(* IEC 61131-3 sources: T4Exjobb/Sigma/Stations/MachineControl/MachineControl/Class/_SysDateTime2, 1 file *)

(* ---- _SysDateTime2.st ---- *)
(*!
<Class
	Name               = "_SysDateTime2"
	Revision           = "0.0"
	RealtimeTask       = "false"
	CyclicTask         = "false"
	BackgroundTask     = "true"
	DefBackground      = "100 ms"
	Sigmatek           = "true"
	OSInterface        = "false"
	HighPriority       = "false"
	Automatic          = "false"
	UpdateMode         = "Prescan"
	SharedCommandTable = "true"
	Objectsize         = "(284,120)">
	<Channels>
		<Server Name="Day" Visualized="true" Initialize="false" WriteProtected="false" Retentive="false"/>
		<Server Name="Hour" Visualized="true" Initialize="false" WriteProtected="false" Retentive="false"/>
		<Server Name="Minute" Visualized="true" Initialize="false" WriteProtected="false" Retentive="false"/>
		<Server Name="Month" Visualized="true" Initialize="false" WriteProtected="false" Retentive="false"/>
		<Server Name="Second" Visualized="true" Initialize="false" WriteProtected="false" Retentive="false"/>
		<Server Name="Year" Visualized="true" Initialize="false" WriteProtected="false" Retentive="false"/>
		<Server Name="Year2Digit" Visualized="true" Initialize="false" WriteProtected="false" Retentive="false"/>
	</Channels>
	<Network Name="_SysDateTime2">
		<!-- List of Components in this network -->
		<Components>
			<Object
				Name           = "_base"
				Class          = "_SysDateTime"
				Position       = "(218,120)"
				Visualized     = "false"
				BackgroundTime = "100 ms">
				<Channels>
					<Server Name="DayOfWeek"/>
					<Server Name="SysDate"/>
					<Server Name="SysTime"/>
					<Client Name="DoSummerTime" Value="0"/>
					<Client Name="System"/>
				</Channels>
			</Object>
		</Components>
		<Comments>
		</Comments>
		<!-- List of Connections in this network -->
		<Connections>
			<Connection Source="this.SysDate" Destination="_base.SysDate" Vertices="(690,210),(518,210),"/>
			<Connection Source="this.SysTime" Destination="_base.SysTime" Vertices="(690,270),(518,270),"/>
			<Connection Source="this.DayOfWeek" Destination="_base.DayOfWeek" Vertices="(690,330),(518,330),"/>
			<Connection Source="_base.System" Destination="this.System" Vertices="(218,210),(38,210),"/>
			<Connection Source="_base.DoSummerTime" Destination="this.DoSummerTime" Vertices="(218,270),(38,270),"/>
		</Connections>
		<!-- Headerfiles -->
		<Options>
		</Options>
	</Network>
</Class>
*)
#pragma using _SysDateTime

_SysDateTime2 : CLASS
: _SysDateTime
  //Servers:
	Second 	: SvrCh_DINT;
	Minute 	: SvrCh_DINT;
	Hour 	: SvrCh_DINT;
	Day 	: SvrCh_DINT;
	Month 	: SvrCh_DINT;
	Year 	: SvrCh_DINT;
	Year2Digit 	: SvrCh_DINT;
  //Clients:
  //Variables:
  //Functions:

	FUNCTION VIRTUAL GLOBAL Background
		VAR_INPUT
			EAX 	: UDINT;
		END_VAR
		VAR_OUTPUT
			state (EAX) 	: UDINT;
		END_VAR;

	FUNCTION VIRTUAL GLOBAL Second::Write
		VAR_INPUT
			input (EAX) 	: DINT;
		END_VAR
		VAR_OUTPUT
			result (EAX) 	: DINT;
		END_VAR;

	FUNCTION VIRTUAL GLOBAL Minute::Write
		VAR_INPUT
			input (EAX) 	: DINT;
		END_VAR
		VAR_OUTPUT
			result (EAX) 	: DINT;
		END_VAR;

	FUNCTION VIRTUAL GLOBAL Hour::Write
		VAR_INPUT
			input (EAX) 	: DINT;
		END_VAR
		VAR_OUTPUT
			result (EAX) 	: DINT;
		END_VAR;

	FUNCTION VIRTUAL GLOBAL Day::Write
		VAR_INPUT
			input (EAX) 	: DINT;
		END_VAR
		VAR_OUTPUT
			result (EAX) 	: DINT;
		END_VAR;

	FUNCTION VIRTUAL GLOBAL Month::Write
		VAR_INPUT
			input (EAX) 	: DINT;
		END_VAR
		VAR_OUTPUT
			result (EAX) 	: DINT;
		END_VAR;

	FUNCTION VIRTUAL GLOBAL Year::Write
		VAR_INPUT
			input (EAX) 	: DINT;
		END_VAR
		VAR_OUTPUT
			result (EAX) 	: DINT;
		END_VAR;

	FUNCTION VIRTUAL GLOBAL Year2Digit::Write
		VAR_INPUT
			input (EAX) 	: DINT;
		END_VAR
		VAR_OUTPUT
			result (EAX) 	: DINT;
		END_VAR;
  //Tables:
	FUNCTION @STD
		VAR_OUTPUT
			ret_code	: CONFSTATES;
		END_VAR;
	FUNCTION GLOBAL TAB @CT_;
END_CLASS;

FUNCTION VIRTUAL GLOBAL _SysDateTime2::Second::Write
	VAR_INPUT
		input (EAX) 	: DINT;
	END_VAR
	VAR_OUTPUT
		result (EAX) 	: DINT;
	END_VAR

  result := ACCESS_DENIED;
  if(SetTimePart(2, to_uint(input)) = true) then
	  Second := input;
 	  result := Second;
  end_if;

END_FUNCTION

FUNCTION VIRTUAL GLOBAL _SysDateTime2::Minute::Write
	VAR_INPUT
		input (EAX) 	: DINT;
	END_VAR
	VAR_OUTPUT
		result (EAX) 	: DINT;
	END_VAR

  result := ACCESS_DENIED;
  if(SetTimePart(1, to_uint(input)) = true) then
	  Minute := input;
 	  result := Minute;
  end_if;

END_FUNCTION

FUNCTION VIRTUAL GLOBAL _SysDateTime2::Hour::Write
	VAR_INPUT
		input (EAX) 	: DINT;
	END_VAR
	VAR_OUTPUT
		result (EAX) 	: DINT;
	END_VAR

  result := ACCESS_DENIED;
  if(SetTimePart(0, to_uint(input)) = true) then
	  Hour := input;
 	  result := Hour;
  end_if;

END_FUNCTION

FUNCTION VIRTUAL GLOBAL _SysDateTime2::Day::Write
	VAR_INPUT
		input (EAX) 	: DINT;
	END_VAR
	VAR_OUTPUT
		result (EAX) 	: DINT;
	END_VAR

  result := ACCESS_DENIED;
  if(SetDatePart(2, to_uint(input)) = true) then
    Day := input;
    result := Day;
  end_if;

END_FUNCTION

FUNCTION VIRTUAL GLOBAL _SysDateTime2::Month::Write
	VAR_INPUT
		input (EAX) 	: DINT;
	END_VAR
	VAR_OUTPUT
		result (EAX) 	: DINT;
	END_VAR

  result := ACCESS_DENIED;
  if(SetDatePart(1, to_uint(input)) = true) then
	  Month := input;
 	  result := Month;
  end_if;

END_FUNCTION

FUNCTION VIRTUAL GLOBAL _SysDateTime2::Year::Write
	VAR_INPUT
		input (EAX) 	: DINT;
	END_VAR
	VAR_OUTPUT
		result (EAX) 	: DINT;
	END_VAR

  result := ACCESS_DENIED;
  if(SetDatePart(0, to_uint(input)) = true) then
	  Year := input;
 	  result := Year;
  end_if;

END_FUNCTION

FUNCTION VIRTUAL GLOBAL _SysDateTime2::Year2Digit::Write
	VAR_INPUT
		input (EAX) 	: DINT;
	END_VAR
	VAR_OUTPUT
		result (EAX) 	: DINT;
	END_VAR
  var
    yy : dint;
  end_var

  if(input < 90) then
    yy := 2000 + input;
  else
    yy := 1900 + input;
  end_if;

  result := Year.Write(yy);

END_FUNCTION

FUNCTION VIRTUAL GLOBAL _SysDateTime2::Background
	VAR_INPUT
		EAX 	: UDINT;
	END_VAR
	VAR_OUTPUT
		state (EAX) 	: UDINT;
	END_VAR

  state := _SysDateTime::Background(eax);

   // HHHHHHHHNNNNNNNNSSSSSSSSxxxxxxxx
  Second := to_dint((SysTime shr  8) and 16#00FF);
  Minute := to_dint((SysTime shr 16) and 16#00FF);
  Hour   := to_dint((SysTime shr 24) and 16#00FF);

  // YYYYYYYYYYYYYYYYMMMMDDDDDDDDWWWW
  Day   := to_dint((SysDate shr  4) and 16#00FF);
  Month := to_dint((SysDate shr 12) and 16#000F);
  Year  := to_dint((SysDate shr 16) and 16#FFFF);

  if(Year >= 2000) then
    Year2Digit := Year - 2000;
  else
    Year2Digit := Year - 1900;
  end_if;

END_FUNCTION
